(* IEC 61131-3 sources: axopen.templates/axopen.template.simple/ax/src/templates/starterunit/Data/_managers_, 3 files *)

(* ---- ProcessDataExchange.st ---- *)
NAMESPACE axosimple.StarterUnitTemplate
    USING axosimple;
    USING AXOpen.Data;
    USING AXOpen.Core;
    USING System.Strings;

    {S7.extern=ReadWrite}
    CLASS ProcessDataExchange
        EXTENDS AXOpen.Data.AxoDataExchange
        VAR PUBLIC
            {#ix-generic:TOnline}
            {#ix-generic:TPlain as POCO}
            {#ix-attr:[AXOpen.Data.AxoDataEntityAttribute]}
            {#ix-attr:[Container(Layout.Stack)]}
            {#ix-set:AttributeName = "<#StarterUnitTemplate#>"}
            Payload : ProcessDataPayload;
        END_VAR
    END_CLASS
END_NAMESPACE

(* ---- TechnologyDataExchange.st ---- *)
NAMESPACE axosimple.StarterUnitTemplate
    USING axosimple;
    USING AXOpen.Data;
    USING AXOpen.Core;
    USING System.Strings;

    {S7.extern=ReadWrite}
    CLASS TechnologyDataExchange
        EXTENDS AXOpen.Data.AxoDataExchange
        VAR PUBLIC
            {#ix-generic:TOnline}
            {#ix-generic:TPlain as POCO}
            {#ix-attr:[AXOpen.Data.AxoDataEntityAttribute]}
            {#ix-attr:[Container(Layout.Stack)]}
            {#ix-set:AttributeName = "<#UnitTemplate#>"}
            Payload : TechnologyDataPayload;
        END_VAR
    END_CLASS
END_NAMESPACE

(* ---- TechnologyDataManager.st ---- *)
NAMESPACE axosimple.StarterUnitTemplate
    USING axosimple;
    USING AXOpen.Data;
    USING AXOpen.Core;
    USING System.Strings;

    {S7.extern=ReadWrite}
    CLASS TechnologyDataManager
        EXTENDS AXOpen.Data.AxoDataFragmentExchange
        VAR PUBLIC
            {#ix-attr:[AXOpen.Data.AxoDataFragmentAttribute]}
            Shared : axosimple.TechnologySharedDataExchange;
            {#ix-attr:[AXOpen.Data.AxoDataFragmentAttribute]}
            Data : TechnologyDataExchange;
        END_VAR
    END_CLASS
END_NAMESPACE
